{attribute 'qualified_only'}
VAR_GLOBAL
	bSwitch1 AT %I*: BOOL;
END_VAR

(* stored: Version 1.1.0.1, ProductVersion 3.1.4024.11
   GVL IO: Id {318c5029-8449-4fc2-b229-5430ffd67ce1} *)
